// TwinCAT 3 PLC project ControlProgram
// ProgramVersion: 3.1.4024.0
// libraries:
//   Tc2_Standard, * (Beckhoff Automation GmbH)
//   Tc2_System, * (Beckhoff Automation GmbH)
//   Tc3_Module, * (Beckhoff Automation GmbH)
// project tree:
//   / PlcTask.TcTTO
//   POUs/ MAIN.TcPOU
// real-time tasks:
//   TASK PlcTask: cycle T#10ms, priority 20, ADS port 350

CONFIGURATION ControlProgram
    RESOURCE PLC ON TwinCAT3
        TASK PlcTask(INTERVAL := T#10ms, PRIORITY := 20);
        PROGRAM MAIN WITH PlcTask : MAIN;
    END_RESOURCE
END_CONFIGURATION

// ---- POUs/MAIN.TcPOU
PROGRAM MAIN
VAR
	Counter :INT;
	i : INT;
	j : INT;
	Timerss :Ton := (IN := TRUE, PT := T#1MS);
	// Michael is a stinker
	// Victor is a real Stinker


END_VAR

//Timerss(IN := TRUE, PT := T#1MS);
Timerss();
Timerss.IN := TRUE;
IF Timerss.Q THEN
	FOR i := 0 TO 100 DO
	Counter := i;

	END_FOR
Timerss.IN := FALSE;

END_IF

END_PROGRAM
